{attribute 'GeneratedUsingTerminal: EL3453-0000-0018'}
{attribute addProperty BoxType "EL3453-0000-0018"}
{attribute addProperty Id "Grid_DirectionAT %I*BOOL1Frequency_Guard_WarningAT %I*BOOL1Frequency_Guard_ErrorAT %I*BOOL1Neutral_Current_Guard_WarningAT %I*BOOL1Neutral_Current_Guard_ErrorAT %I*BOOL1Active_Power_Guard_WarningAT %I*BOOL1Active_Power_Guard_ErrorAT %I*BOOL1Apparent_Power_Guard_WarningAT %I*BOOL1Apparent_Power_Guard_ErrorAT %I*BOOL1Power_Quality_Guard_WarningAT %I*BOOL1Power_Quality_Guard_ErrorAT %I*BOOL1TxPDO_StateAT %I*BOOL1TxPDO_ToggleAT %I*BOOL1Power_Quality_FactorAT %I*REAL4"}
{attribute addProperty CRC "2787890438"}
{attribute addProperty Size "17"}
TYPE Total_Status_A62BD506 :
STRUCT
	{attribute addProperty Name "Grid_Direction"}
	Grid_Direction AT %I* : BOOL;
	{attribute addProperty Name "Frequency_Guard_Warning"}
	Frequency_Guard_Warning AT %I* : BOOL;
	{attribute addProperty Name "Frequency_Guard_Error"}
	Frequency_Guard_Error AT %I* : BOOL;
	{attribute addProperty Name "Neutral_Current_Guard_Warning"}
	Neutral_Current_Guard_Warning AT %I* : BOOL;
	{attribute addProperty Name "Neutral_Current_Guard_Error"}
	Neutral_Current_Guard_Error AT %I* : BOOL;
	{attribute addProperty Name "Active_Power_Guard_Warning"}
	Active_Power_Guard_Warning AT %I* : BOOL;
	{attribute addProperty Name "Active_Power_Guard_Error"}
	Active_Power_Guard_Error AT %I* : BOOL;
	{attribute addProperty Name "Apparent_Power_Guard_Warning"}
	Apparent_Power_Guard_Warning AT %I* : BOOL;
	{attribute addProperty Name "Apparent_Power_Guard_Error"}
	Apparent_Power_Guard_Error AT %I* : BOOL;
	{attribute addProperty Name "Power_Quality_Guard_Warning"}
	Power_Quality_Guard_Warning AT %I* : BOOL;
	{attribute addProperty Name "Power_Quality_Guard_Error"}
	Power_Quality_Guard_Error AT %I* : BOOL;
	{attribute addProperty Name "TxPDO_State"}
	TxPDO_State AT %I* : BOOL;
	{attribute addProperty Name "TxPDO_Toggle"}
	TxPDO_Toggle AT %I* : BOOL;
	{attribute addProperty Name "Power_Quality_Factor"}
	Power_Quality_Factor AT %I* : REAL;
END_STRUCT
END_TYPE

(* stored: Version 1.2.0.0, ProductVersion 3.1.4024.9
   DUT Total_Status_A62BD506: Id {d2e1b99b-27b7-46bf-8547-9d252ad42fc8} *)
